{attribute 'OPC.UA.DA' := '1'}
FUNCTION_BLOCK FB_Sensor_AtlasDO EXTENDS FB_BaseDevice IMPLEMENTS I_Device, I_Sensor

VAR
	
	{attribute 'OPC.UA.DA' := '0'} 
	eSensorType: E_SensorType;
	{attribute 'OPC.UA.DA' := '0'}
	nRawInput AT %I*: INT;
	nFaultInput AT %I*: BOOL;
	{attribute 'OPC.UA.DA' := '1'}
	nCurrentValue: REAL;
	
	{attribute 'OPC.UA.DA' := '0'} 
	nCalOutputLOW AT %Q*: BOOL;
	{attribute 'OPC.UA.DA' := '0'} 
	nCalOutputHIGH AT %Q*: BOOL;
	
	{attribute 'OPC.UA.DA' := '0'} 
	trigCalibrate: R_TRIG;
	
	{attribute 'OPC.UA.DA' := '0'} 
	timerBtnPress: TON := (PT:=T#250MS,IN := FALSE);
	{attribute 'OPC.UA.DA' := '0'} 
	timerDoCalibration: TON := (PT:=T#120S,IN := FALSE); // Check this time during testing! The instructions are not clear about what happens after initiating a calibration request 
	{attribute 'OPC.UA.DA' := '0'} 
	eSMState: (WAIT, LOW_START, LOW_END, HIGH_START, HIGH_END) := WAIT;
	
END_VAR

calculate();
trigCalibrate();
timerBtnPress();


CASE eSMState OF 
	WAIT:
		// wait for the calibrate method call to change the ESMState variable
		

	LOW_START:
		nCalOutputLOW := TRUE;
		timerBtnPress.IN := TRUE;
		IF timerBtnPress.Q THEN
			nCalOutputLOW := FALSE;
			eSMState := LOW_END;
			timerBtnPress.IN := FALSE; 
			timerDoCalibration.IN := TRUE;
		END_IF
		
		eSMState := LOW_END;
		
	LOW_END:
		IF timerDoCalibration.Q THEN
			timerDoCalibration.IN := FALSE;
			bBusy := FALSE;
			eSMState := WAIT;
		END_IF
	
	
	HIGH_START:
		nCalOutputHIGH := TRUE;
		timerBtnPress.IN := TRUE;
		IF timerBtnPress.Q THEN
			nCalOutputHIGH := FALSE;
			eSMState := HIGH_END;
			timerBtnPress.IN := FALSE; 
			timerDoCalibration.IN := TRUE;
		END_IF
		
		eSMState := HIGH_END;
		
	HIGH_END:
		IF timerDoCalibration.Q THEN
			timerDoCalibration.IN := FALSE;
			bBusy := FALSE;
			eSMState := WAIT;
		END_IF
		

END_CASE

METHOD PRIVATE calculate : BOOL
VAR_INPUT
	
	// Var
END_VAR
VAR
	nMeasuredCurrent: REAL;
END_VAR
nMeasuredCurrent := (INT_TO_REAL(nRawInput)/GVL.nMaxADCOutput)*16.0 + 4.0; // in mA


// nCurrentValue := (nMeasuredCurrent - 4.0) * 2.0;  // equation is DO = (mA reading - 4.0) / 0.5

nCurrentValue := (nMeasuredCurrent - 4.0) * 2.0;  // equation is DO = (mA reading - 4.0) / 0.5
END_METHOD

METHOD calibrate : BOOL
VAR_INPUT
	TestType: INT; // LOW = 1, HIGH = 2
END_VAR
CASE TestType OF
	1:
		eSMState := LOW_START;
	2:
		eSMState := HIGH_START;
		
END_CASE

bBusy := TRUE;
END_METHOD

{warning 'add method implementation '}
METHOD disable : BOOL
bEnable := FALSE;
END_METHOD

{warning 'add method implementation '}
METHOD enable : BOOL
bEnable := TRUE;
END_METHOD

{warning 'add method implementation '}
METHOD FB_init : BOOL
VAR_INPUT
	(* if TRUE, the retain variables are initialized (warm start / cold start)*)
	bInitRetains	: BOOL;
	(* if TRUE, the instance afterwards gets moved into the copy code (online change)*)
	bInCopyCode	: BOOL;
	
	SensorID	: STRING(80);
	SensorDescr	: STRING(255);
	SensorType	: E_SensorType;
END_VAR
sID := SensorID;
sDescr := SensorDescr;
eSensorType := SensorType;
END_METHOD

{warning 'add method implementation '}
METHOD getType : E_SensorType
getType := eSensorType;
END_METHOD

{warning 'add method implementation '}
METHOD getValue : REAL
getValue := nCurrentValue;
END_METHOD

{warning 'add method implementation '}
METHOD write : BOOL
// use this method to initiated a hardware read from assigned IO if required
END_METHOD

END_FUNCTION_BLOCK

(* stored: Version 1.1.0.1, ProductVersion 3.1.4024.12
   POU FB_Sensor_AtlasDO: Id {311373c6-d3a1-46f8-8bbf-36579a150e3d}, SpecialFunc None
   Method calculate: Id {aa77c180-02ca-4169-8e47-9f714ed550a6}
   Method calibrate: Id {3bbf9354-c59b-42d4-9aa6-4f5a4fe072f9}
   Method disable: Id {b56074bd-5d3d-4815-b679-163f0a6343f7}
   Method enable: Id {75fbd39c-834d-401b-85ca-55cdda0e7f23}
   Method FB_init: Id {ac500d8b-f0e9-4c01-b5cd-3b9100ee7394}
   Method getType: Id {cb0bdbee-0271-4d1b-bd59-9fea4b1f33db}
   Method getValue: Id {f1da22c0-9dd5-4237-85d8-d4d3b383fc16}
   Method write: Id {46b1587a-c6ed-4aff-adc8-c4ceeb3ef79a} *)
